// TIA Portal V16 export
// export: Created 2021-07-12T14:47:15.2802004Z, ExportSetting WithDefaults, DisplayName Totally Integrated Automation Portal, DisplayVersion V16, DisplayName TIA Portal Version Control Interface, DisplayVersion V16, DisplayName TIA Portal Openness, DisplayVersion V16, DisplayName STEP 7 Professional, DisplayVersion V16, DisplayName STEP 7 Safety, DisplayVersion V16, DisplayName WinCC Professional, DisplayVersion V16
DATA_BLOCK "InstSimaHydTO_HMI"   // DB33105
TITLE = InstSimaHydTO_HMI
{ DB_Accessible_From_OPC_UA := 'FALSE' }
FAMILY : SimaHydTO
VERSION : 1.0
// Instance data block
// stored: AutoNumber true, DBAccessibleFromOPCUA false, InstanceOfName SimaHydTO_HMI, InstanceOfType FB
"SimaHydTO_HMI"
   // VAR_IN_OUT
   //    hmiConnection : "SimaHydTO_typeHMIConnection";
   //    axesArray : Array[*] of "SimaHydTO_typeAxesArray";
   //    vCharArray : Array[*] of "SimaHydTO_typeVCharArray";
   // END_VAR
   // VAR
   //    statInitObjects { ExternalAccessible := 'False'; ExternalVisible := 'False'; ExternalWritable := 'False'} : Bool;
   //    instHmiAxisSelector { ExternalAccessible := 'False'; ExternalVisible := 'False'; ExternalWritable := 'False'; S7_SetPoint := 'True'} : "SimaHydTO_HmiAxisSelector";
   //    instHmiVCharSelector { ExternalAccessible := 'False'; ExternalVisible := 'False'; ExternalWritable := 'False'; S7_SetPoint := 'True'} : "SimaHydTO_HmiVCharSelector";
   //    instBasicAxisControl { ExternalAccessible := 'False'; ExternalVisible := 'False'; ExternalWritable := 'False'; S7_SetPoint := 'True'} : "SimaHydTO_BasicAxisControl";
   //    instVCharMeasurement { ExternalAccessible := 'False'; ExternalVisible := 'False'; ExternalWritable := 'False'; S7_SetPoint := 'True'} : "SimaHydTO_VCharMeasurement";
   //    instVCharEditor { ExternalAccessible := 'False'; ExternalVisible := 'False'; ExternalWritable := 'False'; S7_SetPoint := 'True'} : "SimaHydTO_VCharEditor";
   //    instAdvancedAxisControl { ExternalAccessible := 'False'; ExternalVisible := 'False'; ExternalWritable := 'False'; S7_SetPoint := 'True'} : "SimaHydTO_AdvancedAxisControl";
   //    instParameterSettings { ExternalAccessible := 'False'; ExternalVisible := 'False'; ExternalWritable := 'False'; S7_SetPoint := 'True'} : "SimaHydTO_ParameterSettings";
   //    instFindVChars { ExternalAccessible := 'False'; ExternalVisible := 'False'; ExternalWritable := 'False'; S7_SetPoint := 'True'} : "SimaHydTO_FindObjects";
   //    instVCharManagement { ExternalAccessible := 'False'; ExternalVisible := 'False'; ExternalWritable := 'False'; S7_SetPoint := 'True'} : "SimaHydTO_VCharManagement";
   // END_VAR
BEGIN
END_DATA_BLOCK
